(* IEC 61131-3 sources: RAG_PLC/data/result/test/050, 2 files *)

(* ---- wrapped.st ---- *)
(* =========================================================
   Generated by PLC-Eval Benchmark Wrapper
   ========================================================= *)

FUNCTION_BLOCK LLM_Wrapper_FB
VAR_INPUT
    X : REAL;
END_VAR

VAR_OUTPUT
    FRACT : REAL;
END_VAR

IF ABS(X) < 2.0E9 THEN
    FRACT := X - DINT_TO_REAL(D_TRUNC(X));
ELSE
    FRACT := 0.0;
END_IF;
END_FUNCTION_BLOCK

PROGRAM Auto_Proxy_Prg
  VAR
    instance : LLM_Wrapper_FB;
  END_VAR

  instance();
END_PROGRAM

CONFIGURATION Config0
  RESOURCE Res0 ON PLC
    TASK TaskMain(INTERVAL := T#20ms, PRIORITY := 0);
    PROGRAM Inst0 WITH TaskMain : Auto_Proxy_Prg;
  END_RESOURCE
END_CONFIGURATION

(* ---- raw_code.st ---- *)
VAR_INPUT
    X : REAL;
END_VAR

VAR_OUTPUT
    FRACT : REAL;
END_VAR

IF ABS(X) < 2.0E9 THEN
    FRACT := X - DINT_TO_REAL(D_TRUNC(X));
ELSE
    FRACT := 0.0;
END_IF;
